{attribute 'qualified_only'}
{attribute 'strict'}
{attribute 'to_string'}
TYPE SidesMaterialsEnum :
(
	//CARDBOARD
	CAR20S, CAR20M, CAR20L, CAR28S, CAR28M, CAR28L, //base (flat)
	
	//CHIPBOARD
	CIP18, CIP54,
	
	//WOOD BUNK
	WDS08, WDS10, WDS12, WDS14, WDS20, WDS22, WDS28, //side
	WDS8X8, WDS8X10, WDS12X12, WDS12X14, WDS20X10, WDS20X12, //side combined - X
	
	size //number of materials
);
END_TYPE

(* stored: Version 1.1.0.1, ProductVersion 3.1.4024.11
   EnumerationTextList SidesMaterialsEnum: Id {1de8278d-b6a6-4aea-b779-a0d856b091a1} *)
